{attribute 'GeneratedUsingTerminal: EL4032-0000-0016'}
{attribute addProperty BoxType "EL4032-0000-0016"}
{attribute addProperty Description "EL4032 2Ch. Ana. Output +/-10V, 12bit"}
{attribute addProperty Physics "KK"}
{attribute addProperty Id "AO_Outputs_Channel_1AT %Q*AO_Output_Channel_BA7EBB7C2AO_Outputs_Channel_2AT %Q*AO_Output_Channel_BA7EBB7C2WcStateAT %I*WcState_0B2B16F91InfoDataAT %I*InfoData_32EB74EA10"}
{attribute addProperty CRC "300123737"}
{attribute addProperty Size "15"}
TYPE EL4032_11E38659 EXTENDS EtcSlaveTerminalBase_947E5A46 :
STRUCT
	{attribute addProperty Name "AO_Outputs_Channel_1"}
	AO_Outputs_Channel_1 : AO_Output_Channel_BA7EBB7C;
	{attribute addProperty Name "AO_Outputs_Channel_2"}
	AO_Outputs_Channel_2 : AO_Output_Channel_BA7EBB7C;
	{attribute addProperty Name "WcState"}
	WcState : WcState_0B2B16F9;
	{attribute addProperty Name "InfoData"}
	InfoData : InfoData_32EB74EA;
END_STRUCT
END_TYPE

(* stored: Version 1.2.0.0, ProductVersion 3.1.4024.9
   DUT EL4032_11E38659: Id {c83d284a-7e9b-4fd7-8ee8-a06fd73b971a} *)
